PROGRAM MAIN
VAR	

END_VAR

// GVL Variable For Prep
GVL.HMI_Prep_Name_Display[0] := 'Test';
GVL.HMI_Prep_Name_Display[1] := 'Test';
GVL.HMI_Prep_Name_Display[2] := 'Test';
GVL.HMI_Prep_Name_Display[3] := 'Test';
GVL.HMI_Prep_Name_Display[4] := 'Test';
GVL.HMI_Prep_Name_Display[5] := 'Test';
GVL.HMI_Prep_Name_Display[6] := 'Test';
GVL.HMI_Prep_Name_Display[7] := 'Test';

GVL.HMI_Prep_Name_Input[0] := 'Test';
GVL.HMI_Prep_Name_Input[1] := 'Test';
GVL.HMI_Prep_Name_Input[2] := 'Test';
GVL.HMI_Prep_Name_Input[3] := 'Test';

GVL.HMI_Prep_Name_IO[0] := 'Test';
GVL.HMI_Prep_Name_IO[1] := 'Test';
GVL.HMI_Prep_Name_IO[2] := 'Test';
GVL.HMI_Prep_Name_IO[3] := 'Test';

END_PROGRAM

(* stored: Version 1.1.0.1, ProductVersion 3.1.4024.12
   POU MAIN: Id {3aac644e-6292-47e0-b79d-c2fce7bfcc53}, SpecialFunc None *)
